FUNCTION_BLOCK AnalogicalSwitch (* Basic FB with empty ECC *)
  (* Standard: 61499-2 *)
  (* Version 1.0, 2021-12-09, Fan *)
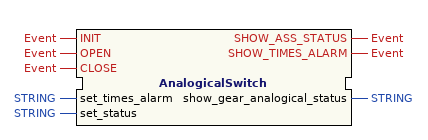
  EVENT_INPUT
    INIT; (* Initialise the Open and Close at the event *)
    OPEN; (* Event tick Open message  when pilot press the button *)
    CLOSE; (* Event tick Open message  when pilot press the button *)
  END_EVENT
  EVENT_OUTPUT
    SHOW_ASS_STATUS;
    SHOW_TIMES_ALARM;
  END_EVENT
  VAR_INPUT
    set_times_alarm : STRING; (* Static input paramter to set the alarm *)
    set_status : STRING; (* status get from gear lever *)
  END_VAR
  VAR_OUTPUT
    show_gear_analogical_status : STRING; (* Final status display *)
  END_VAR
  EC_STATES
    START; (* Initial State *)
  END_STATES
END_FUNCTION_BLOCK
